Fanuc TP program (LS listing): _PICK_ARRAY.LS

/PROG  _PICK_ARRAY
/ATTR
OWNER		= MNEDITOR;
COMMENT		= "Pick SubRoutine";
PROG_SIZE	= 1812;
CREATE		= DATE 22-08-19  TIME 15:17:30;
MODIFIED	= DATE 23-12-13  TIME 09:54:20;
FILE_NAME	= ;
VERSION		= 0;
LINE_COUNT	= 57;
MEMORY_SIZE	= 2216;
PROTECT		= READ_WRITE;
TCD:  STACK_SIZE	= 0,
      TASK_PRIORITY	= 50,
      TIME_SLICE	= 0,
      BUSY_LAMP_OFF	= 0,
      ABORT_REQUEST	= 0,
      PAUSE_REQUEST	= 7;
DEFAULT_GROUP	= 1,*,*,*,*;
CONTROL_CODE	= 00000000 00000000;
LOCAL_REGISTERS	= 0,0,0;
/APPL
/APPL

AUTO_SINGULARITY_HEADER;
  ENABLE_SINGULARITY_AVOIDANCE   : TRUE;
/MN
   1:  !************************ ;
   2:  ! Example of Part Array ;
   3:  ! Use any UT and UF     ;
   4:  !************************ ;
   5:  UFRAME_NUM=9 ;
   6:  UTOOL_NUM=1 ;
   7:   ;
   8:  !Init Registers ;
   9:  R[130:LayerIndex]=0    ;
  10:  R[131:CurrentColumn;]=0    ;
  11:  R[132:CurrentRow;]=0    ;
  12:  PR[99:TempPR]=LPOS-LPOS    ;
  13:   ;
  14:  !Set Total Parts ;
  15:  R[133:TotalParts]=R[135:MaxColumns]*R[136:MaxRows]    ;
  16:   ;
  17:  !------------------- ;
  18:  LBL[10:Start] ;
  19:  !------------------- ;
  20:  PAUSE ;
  21:  ! Pick Part               ;
  22:  !  current row =          ;
  23:  !   index MOD max columns ;
  24:  R[132:CurrentRow]=R[130:LayerIndex] MOD R[135:MaxColumns]    ;
  25:   ;
  26:  ! current col = ;
  27:  ! index DIV  max columns ;
  28:  R[131:CurrentColumn]=R[130:LayerIndex] DIV R[135:MaxColumns]    ;
  29:   ;
  30:  ! Set offset X and Y             ;
  31:  !  current column =              ;
  32:  !   curr column * column offset  ;
  33:  R[131:CurrentColumn]=R[131:CurrentColumn]*R[137:ColumnOffset]    ;
  34:   ;
  35:  ! current row =          ;
  36:  !  curr row * row offset ;
  37:  R[132:CurrentRow]=R[132:CurrentRow;]*R[138:RowOffset;]    ;
  38:   ;
  39:  ! Apply offset X and Y ;
  40:  PR[99,1]=R[132:CurrentRow;]    ;
  41:  PR[99,2]=R[131:CurrentColumn;]    ;
  42:  ! Use taugh pos with      ;
  43:  !  updated PR for Offset ;
  44:J P[2:PickPt] 100% FINE Offset,PR[99]    ;
  45:   ;
  46:  ! Increment Index Counter ;
  47:  R[130:LayerIndex]=R[130:LayerIndex]+1    ;
  48:   ;
  49:  ! Total Parts sets loop counter ;
  50:  IF R[130:LayerIndex]<R[133:TotalParts],JMP LBL[10] ;
  51:   ;
  52:  END ;
  53:  !-------------------- ;
  54:  !  Touchup            ;
  55:  !-------------------- ;
  56:J P[2:PickPt] 100% FINE    ;
  57:   ;
/POS
P[2:"PickPt"]{
   GP1:
	UF : 9, UT : 1,		CONFIG : 'F U T, 0, 0, 0',
	X =   144.121262  mm,	Y =   138.303909  mm,	Z =     2.001340  mm,
	W =   178.737549 deg,	P =     -.681968 deg,	R =  -179.327591 deg
};
/END
